% RSLogix 500 project PROC1_SEGREGATING_IO_BAK001.RSS, saved by version 8.30.00.16 %
PROJECT "PROC1"    % processor: Bul.1763 MicroLogix 1100 Series B %

PROGRAM FILES
  LAD 2 "MAIN"  2 rungs
  LAD 3 "IO"  3 rungs

DATA FILES
  O0 OUTPUT  5 elements
  I1 INPUT  7 elements
  S2 STATUS  66 elements
  B3 BINARY  1 elements
  T4 TIMER  1 elements
  C5 COUNTER  1 elements
  R6 CONTROL  1 elements
  N7 INTEGER  1 elements
  F8 FLOAT  1 elements

LADDER 2 "MAIN"
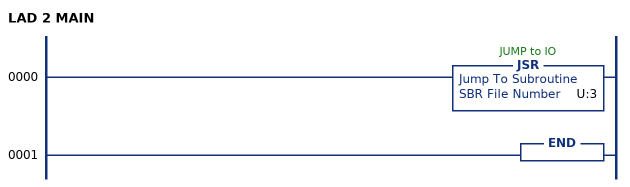
% Rung: 0 %
SOR JSR U:3 EOR
%   U:3  "JUMP to IO" %
% Rung: 1 %
SOR END EOR

LADDER 3 "IO"
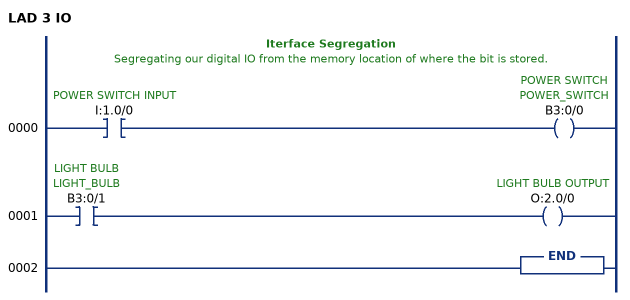
% Rung: 0 %
% TITLE: Iterface Segregation %
% Segregating our digital IO from the memory location of where the bit is stored. %
SOR XIC I:1.0/0 OTE B3:0/0 EOR
%   I:1.0/0  "POWER SWITCH INPUT" %
%   B3:0/0  POWER_SWITCH  "POWER SWITCH" %
% Rung: 1 %
SOR XIC B3:0/1 OTE O:2.0/0 EOR
%   B3:0/1  LIGHT_BULB  "LIGHT BULB" %
%   O:2.0/0  "LIGHT BULB OUTPUT" %
% Rung: 2 %
SOR END EOR

REVISION NOTES
  0: Added IO rungs
